// TIA Portal V19 export
FUNCTION_BLOCK "HU_Tank"   // FB107, LAD
TITLE = Hydraulic Tank Machine / HYDRAULIC UNIT (MONO-PUMP)
// stored: Access Published, MemoryReserve 100, SetENOAutomatically false
   VAR_INPUT
      AreaInterface : "AreaInterface";
      DataIn : Struct
         SensorLevelOk_Warning : Bool;
         SensorLevelOk_Alarm : Bool;
         SensorOilMaxTempOk : Bool;
         SensorRecircFilterClogged : Bool;
         SwThermostatCooling : Bool;
         RecircPump_FdbkRunning : Bool;
         HeatExchangeFan_FdbkRunning : Bool;
         HeatingUnit1_FdbkRunning : Bool;
         HeatingUnit2_FdbkRunning : Bool;
         ChillerWaterFluxOk : Bool;
         ChillerAlarmPresence : Bool;
         Anl_OilTemperature : Int;
         Anl_WaterTemperature : Int;
      END_STRUCT;
      CIn : Struct
         PumpRunning : Bool;   // From HU_Pump
      END_STRUCT;
      Config : "HU_Tank_Config";
      Simulation : Bool;
   END_VAR
   VAR_OUTPUT
      MachineInterface : "MachineInterface";
      DataOut : Struct
         KmHeatExchangerFan : Bool;
         KmRecirculationPump : Bool;
         KmHeatingUnit1 : Bool;
         KmHeatingUnit2 : Bool;
         EvChillerWater : Bool;
      END_STRUCT;
      COut : Struct
         PumpRunPermitted : Bool;   // For HU_Pump
         EnableCheckFIler : Bool;   // For HU_Pump
      END_STRUCT;
   END_VAR
   VAR_IN_OUT
      Par : "HU_Tank_Par";
   END_VAR
   VAR
      M_RecirculationPump : "Motor";
      M_HeatExchangerFan : "Motor";
      M_HeatingUnit1 : "Motor";
      M_HeatingUnit2 : "Motor";
      Ctrl : Struct
         RstAlarms : Bool;
         RecirculationPump_Run : Bool;
         HeatExchangerFan_Run : Bool;
         HeatingUnit1_Run : Bool;
         HeatingUnit2_Run : Bool;
      END_STRUCT;
      Sts : Struct
         AlarmsPresence : Bool;
         WarningsPresence : Bool;
         IsStandstill : Bool;
         CoolingReq : Bool;
         HeatingReq : Bool;
         CndRecirculationPump : Bool;
         CndHeatExchangerFan : Bool;
         CndHeatingUnit : Bool;
         OilMaxTemperature : Bool;
         FilterWatchEnableByTemperature : Bool;
         WeeklyClockEnabled : Bool;
         OilTemperature : Real;
         WaterTemperature : Real;
      END_STRUCT;
      HMI : "HU_Tank_HMI";
      Alarm : Struct
         LowTankLevel : Bool;
         OilMaxTemperature : Bool;
         RecircFilterClogged : Bool;
         RecirculationPump : "MotorAlr";
         HeatExchangerFan : "MotorAlr";
         HeatingUnit1 : "MotorAlr";
         HeatingUnit2 : "MotorAlr";
      END_STRUCT;
      Warning : Struct
         NoAutReady : Bool;
         LowTankLevel : Bool;
         CoolingActive : Bool;
         HeatingActive : Bool;
         ChillerLowWater : Bool;
         ChillerAlarm : Bool;
         ChillerWaterMaxTemp : Bool;
         WaitingStartCondition : Bool;
      END_STRUCT;
      tonLowLevel_Warning : IEC_TIMER;
      tonLowLevel_Alarm : IEC_TIMER;
      tonOilMaxTemperature : IEC_TIMER;
      tonAlrRecircFilterClogged : IEC_TIMER;
      tonRecirculationPumpStop : IEC_TIMER;
      tonCoolingStop : IEC_TIMER;
      tonCoolingStart : IEC_TIMER;
      tonDelayCheckChiller : IEC_TIMER;
      tonDelayStartHeating1 : IEC_TIMER;
      tonDelayStopHeating1 : IEC_TIMER;
      tonDelayStartHeating2 : IEC_TIMER;
      tonDelayStopHeating2 : IEC_TIMER;
   END_VAR
   VAR DB_SPECIFIC
      ActualDT : DTL;
      ActualDate : Date;
      ActuaDtON : DTL;
      ActualDtOFF : DTL;
   END_VAR
   VAR
      AckRstAlarms : Bool;
   END_VAR
   VAR_TEMP
      ScaleRetVal : Word;
      StartHeating : Real;
      StopHeating : Real;
      DateRetVal : Int;
      IsGt : Bool;
      IsLt : Bool;
   END_VAR
BEGIN

REGION Network 1 (SCL): Info
   //=============================================================================
   //PM FORMING
   //-----------------------------------------------------------------------------
   // Library: StandardBlocks
   // Tested with: S7-1518TF
   // Engineering: TIA Portal V18
   // Restrictions: -
   // Requirements: S7-1500
   // Functionality: Hydraulic Tank Machine
   //
   // v1.0.0  28/12/2022 
   // v1.0.1  16/01/2023 Added Weekly clock
   // v1.1.0  14/02/2023 Simulation added
   // v1.1.1  11/05/2023 Added config analogic High and low limit
   // v1.1.2  14/06/2023 Set Sensor filter clogged NO
   // v1.1.3  13/11/2023 Add recirculation pump not exist for heating condition
   // v1.1.4  05/03/2024 Add condition low level for recirculation and heating unit
   // v1.1.5  29/04/2024 Add reset filter clogged
   //=============================================================================
END_REGION

REGION Network 2 (SCL): Reset alarms command
   #Ctrl.RstAlarms := #AreaInterface.RstAlarms AND NOT #AckRstAlarms;
   #AckRstAlarms := #AreaInterface.RstAlarms;

   IF #Ctrl.RstAlarms THEN
       #Warning.NoAutReady := FALSE;
       #Alarm.LowTankLevel :=  FALSE;
       #Alarm.OilMaxTemperature := FALSE;    
       #Alarm.RecircFilterClogged := FALSE;
   END_IF;
END_REGION

REGION Network 3: Warning low level
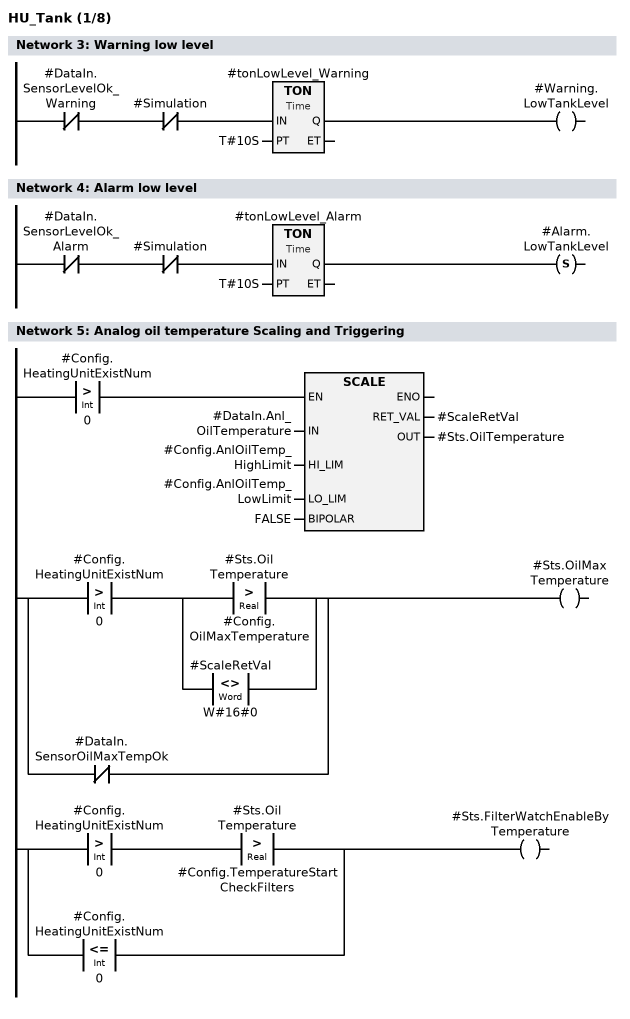
   RUNG wire#powerrail
      I_Contact( #DataIn.SensorLevelOk_Warning )
      I_Contact( #Simulation )
      { S7_Templates := "time_type := Time" } #tonLowLevel_Warning.TON(pt := T#10S, et =>)
      Coil( #Warning.LowTankLevel )
   END_RUNG
   // the same network as SCL:
   #tonLowLevel_Warning.TON(IN := NOT #DataIn.SensorLevelOk_Warning AND NOT #Simulation, PT := T#10S);
   #Warning.LowTankLevel := #tonLowLevel_Warning.Q;
END_REGION

REGION Network 4: Alarm low level
   RUNG wire#powerrail
      I_Contact( #DataIn.SensorLevelOk_Alarm )
      I_Contact( #Simulation )
      { S7_Templates := "time_type := Time" } #tonLowLevel_Alarm.TON(pt := T#10S, et =>)
      S_Coil( #Alarm.LowTankLevel )
   END_RUNG
   // the same network as SCL:
   #tonLowLevel_Alarm.TON(IN := NOT #DataIn.SensorLevelOk_Alarm AND NOT #Simulation, PT := T#10S);
   IF #tonLowLevel_Alarm.Q THEN #Alarm.LowTankLevel := TRUE; END_IF;
END_REGION

REGION Network 5: Analog oil temperature Scaling and Triggering
   IF #Config.HeatingUnitExistNum > 0 THEN
       #ScaleRetVal := SCALE(IN := #DataIn.Anl_OilTemperature,
                             HI_LIM := #Config.AnlOilTemp_HighLimit,
                             LO_LIM := #Config.AnlOilTemp_LowLimit,
                             BIPOLAR := FALSE,
                             OUT => #Sts.OilTemperature);
   END_IF;
   #Sts.OilMaxTemperature := ((#Config.HeatingUnitExistNum > 0) AND ((#Sts.OilTemperature > #Config.OilMaxTemperature) OR (#ScaleRetVal <> W#16#0))) OR NOT #DataIn.SensorOilMaxTempOk;
   #Sts.FilterWatchEnableByTemperature := ((#Config.HeatingUnitExistNum > 0) AND (#Sts.OilTemperature > #Config.TemperatureStartCheckFilters)) OR (#Config.HeatingUnitExistNum <= 0);
END_REGION

REGION Network 6: Analog water temperature Scaling and Triggering
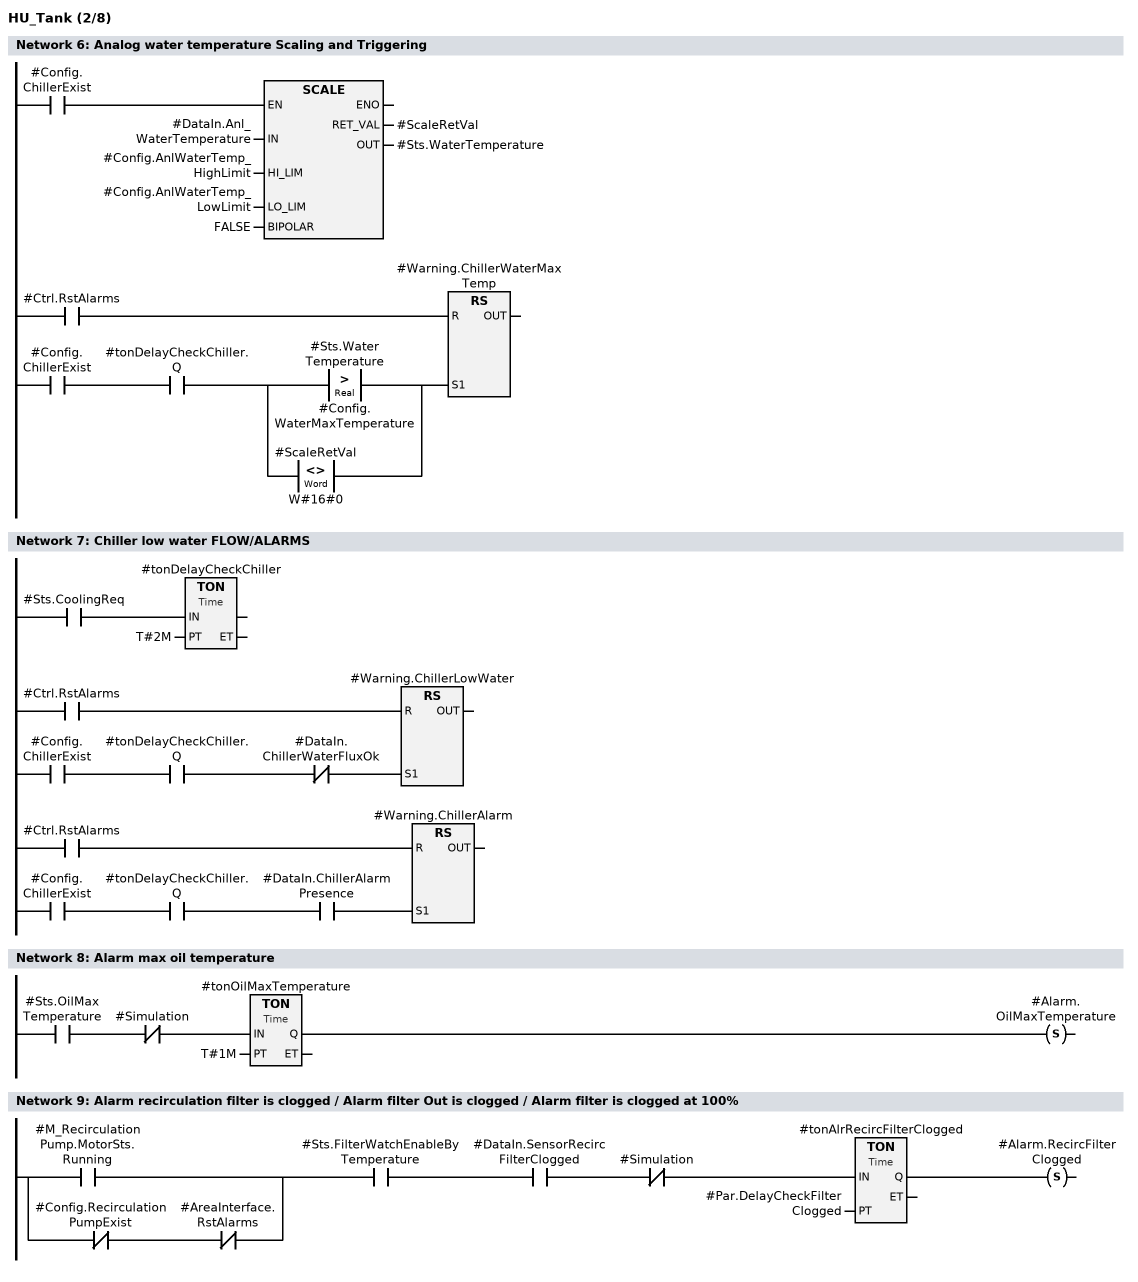
   IF #Config.ChillerExist THEN
       #ScaleRetVal := SCALE(IN := #DataIn.Anl_WaterTemperature,
                             HI_LIM := #Config.AnlWaterTemp_HighLimit,
                             LO_LIM := #Config.AnlWaterTemp_LowLimit,
                             BIPOLAR := FALSE,
                             OUT => #Sts.WaterTemperature);
   END_IF;
   IF #Ctrl.RstAlarms THEN
       #Warning.ChillerWaterMaxTemp := FALSE;   // RS flip-flop
   END_IF;
   IF #Config.ChillerExist AND #tonDelayCheckChiller.Q AND ((#Sts.WaterTemperature > #Config.WaterMaxTemperature) OR (#ScaleRetVal <> W#16#0)) THEN
       #Warning.ChillerWaterMaxTemp := TRUE;
   END_IF;
END_REGION

REGION Network 7: Chiller low water FLOW/ALARMS
   RUNG wire#powerrail
      Contact( #Sts.CoolingReq )
      { S7_Templates := "time_type := Time" } #tonDelayCheckChiller.TON(pt := T#2M, et =>)
   END_RUNG
   RUNG wire#powerrail
      Contact( #Ctrl.RstAlarms )
      S_RS(operand := #Warning.ChillerLowWater, s1 := wire#w1)
   END_RUNG
   RUNG wire#powerrail
      Contact( #Config.ChillerExist )
      Contact( #tonDelayCheckChiller.Q )
      I_Contact( #DataIn.ChillerWaterFluxOk )
   END_RUNG wire#w1
   RUNG wire#powerrail
      Contact( #Ctrl.RstAlarms )
      S_RS(operand := #Warning.ChillerAlarm, s1 := wire#w2)
   END_RUNG
   RUNG wire#powerrail
      Contact( #Config.ChillerExist )
      Contact( #tonDelayCheckChiller.Q )
      Contact( #DataIn.ChillerAlarmPresence )
   END_RUNG wire#w2
   // the same network as SCL:
   #tonDelayCheckChiller.TON(IN := #Sts.CoolingReq, PT := T#2M);
   IF #Ctrl.RstAlarms THEN
       #Warning.ChillerLowWater := FALSE;   // RS flip-flop
   END_IF;
   IF #Config.ChillerExist AND #tonDelayCheckChiller.Q AND NOT #DataIn.ChillerWaterFluxOk THEN
       #Warning.ChillerLowWater := TRUE;
   END_IF;
   IF #Ctrl.RstAlarms THEN
       #Warning.ChillerAlarm := FALSE;   // RS flip-flop
   END_IF;
   IF #Config.ChillerExist AND #tonDelayCheckChiller.Q AND #DataIn.ChillerAlarmPresence THEN
       #Warning.ChillerAlarm := TRUE;
   END_IF;
END_REGION

REGION Network 8: Alarm max oil temperature
   RUNG wire#powerrail
      Contact( #Sts.OilMaxTemperature )
      I_Contact( #Simulation )
      { S7_Templates := "time_type := Time" } #tonOilMaxTemperature.TON(pt := T#1M, et =>)
      S_Coil( #Alarm.OilMaxTemperature )
   END_RUNG
   // the same network as SCL:
   #tonOilMaxTemperature.TON(IN := #Sts.OilMaxTemperature AND NOT #Simulation, PT := T#1M);
   IF #tonOilMaxTemperature.Q THEN #Alarm.OilMaxTemperature := TRUE; END_IF;
END_REGION

REGION Network 9: Alarm recirculation filter is clogged / Alarm filter Out is clogged / Alarm filter is clogged at 100%
   RUNG wire#powerrail
      Contact( #M_RecirculationPump.MotorSts.Running )
      wire#w1
      Contact( #Sts.FilterWatchEnableByTemperature )
      Contact( #DataIn.SensorRecircFilterClogged )
      I_Contact( #Simulation )
      { S7_Templates := "time_type := Time" } #tonAlrRecircFilterClogged.TON(pt := #Par.DelayCheckFilterClogged, et =>)
      S_Coil( #Alarm.RecircFilterClogged )
   END_RUNG
   RUNG wire#powerrail
      I_Contact( #Config.RecirculationPumpExist )
      I_Contact( #AreaInterface.RstAlarms )
   END_RUNG wire#w1
   // the same network as SCL:
   #tonAlrRecircFilterClogged.TON(IN := (#M_RecirculationPump.MotorSts.Running OR (NOT #Config.RecirculationPumpExist AND NOT #AreaInterface.RstAlarms)) AND #Sts.FilterWatchEnableByTemperature AND #DataIn.SensorRecircFilterClogged AND NOT #Simulation,
                           PT := #Par.DelayCheckFilterClogged);
   IF #tonAlrRecircFilterClogged.Q THEN #Alarm.RecircFilterClogged := TRUE; END_IF;
END_REGION

REGION Network 11: <<< HEAT EXCHANGER (RECIRCULATION PUMP & COOLING FAN) / <<< RECIRCULATION PUMP & COOLING FAN >>>
END_REGION

REGION Network 12: Main / Cooling request / Cooling request by thermostat
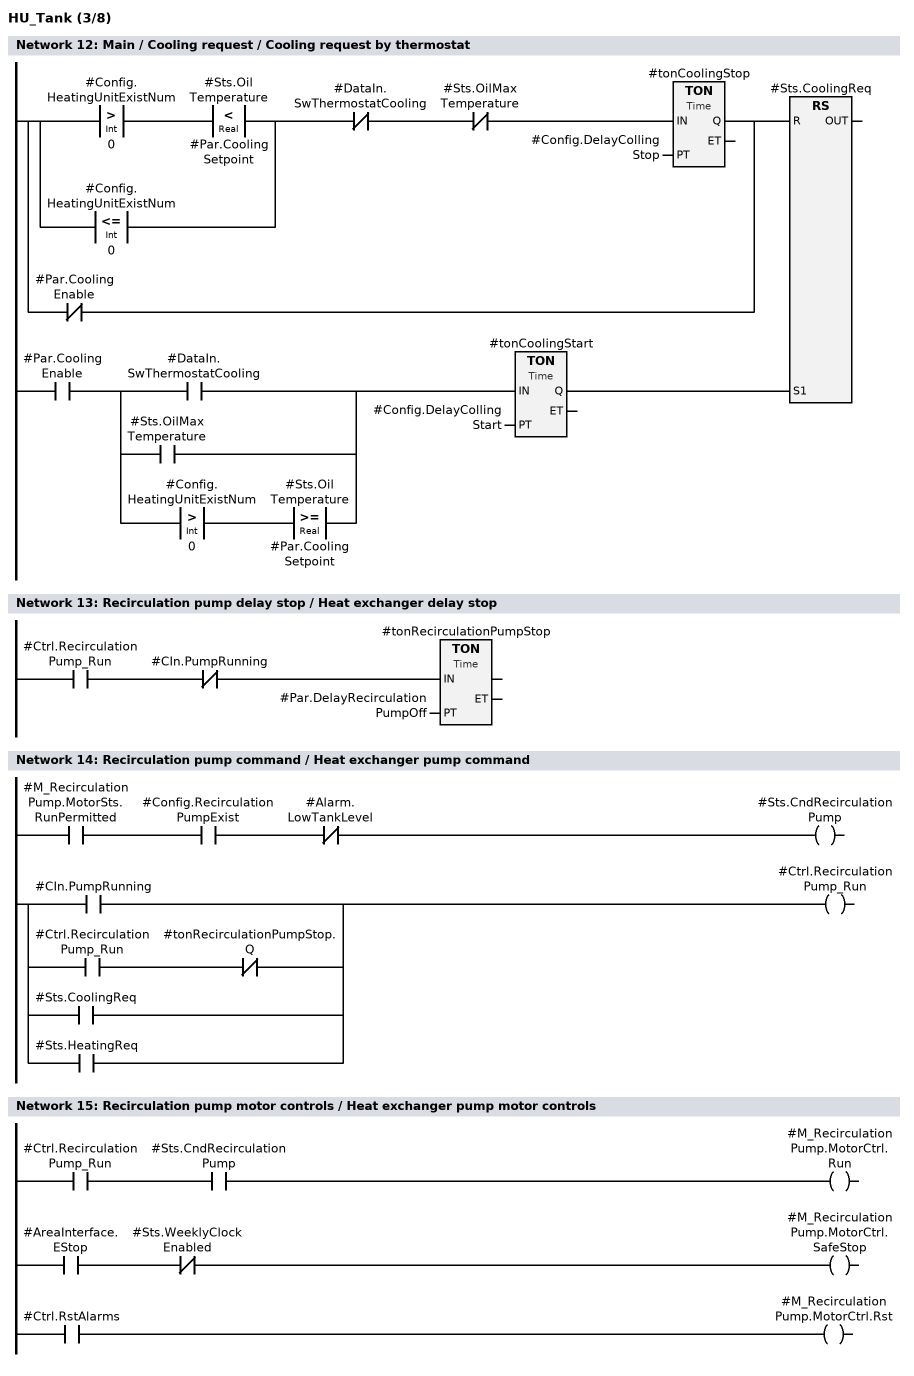
   RUNG wire#powerrail
      { S7_Templates := "SrcType := Int" } GT_Contact(in1 := #Config.HeatingUnitExistNum, in2 := 0)
      { S7_Templates := "SrcType := Real" } LT_Contact(in1 := #Sts.OilTemperature, in2 := #Par.CoolingSetpoint)
      wire#w1
      I_Contact( #DataIn.SwThermostatCooling )
      I_Contact( #Sts.OilMaxTemperature )
      { S7_Templates := "time_type := Time" } #tonCoolingStop.TON(pt := #Config.DelayCollingStop, et =>)
      wire#w2
      S_RS(operand := #Sts.CoolingReq, s1 := wire#w5)
   END_RUNG
   RUNG wire#powerrail
      { S7_Templates := "SrcType := Int" } LE_Contact(in1 := #Config.HeatingUnitExistNum, in2 := 0)
   END_RUNG wire#w1
   RUNG wire#powerrail
      I_Contact( #Par.CoolingEnable )
   END_RUNG wire#w2
   RUNG wire#powerrail
      Contact( #Par.CoolingEnable )
      wire#w3
      Contact( #DataIn.SwThermostatCooling )
      wire#w4
      { S7_Templates := "time_type := Time" } #tonCoolingStart.TON(pt := #Config.DelayCollingStart, et =>)
   END_RUNG wire#w5
   RUNG wire#w3
      Contact( #Sts.OilMaxTemperature )
   END_RUNG wire#w4
   RUNG wire#w3
      { S7_Templates := "SrcType := Int" } GT_Contact(in1 := #Config.HeatingUnitExistNum, in2 := 0)
      { S7_Templates := "SrcType := Real" } GE_Contact(in1 := #Sts.OilTemperature, in2 := #Par.CoolingSetpoint)
   END_RUNG wire#w4
   // the same network as SCL:
   #tonCoolingStop.TON(IN := (((#Config.HeatingUnitExistNum > 0) AND (#Sts.OilTemperature < #Par.CoolingSetpoint)) OR (#Config.HeatingUnitExistNum <= 0)) AND NOT #DataIn.SwThermostatCooling AND NOT #Sts.OilMaxTemperature,
                       PT := #Config.DelayCollingStop);
   #tonCoolingStart.TON(IN := #Par.CoolingEnable AND (#DataIn.SwThermostatCooling OR #Sts.OilMaxTemperature OR ((#Config.HeatingUnitExistNum > 0) AND (#Sts.OilTemperature >= #Par.CoolingSetpoint))),
                        PT := #Config.DelayCollingStart);
   IF #tonCoolingStop.Q OR NOT #Par.CoolingEnable THEN
       #Sts.CoolingReq := FALSE;   // RS flip-flop
   END_IF;
   IF #tonCoolingStart.Q THEN #Sts.CoolingReq := TRUE; END_IF;
END_REGION

REGION Network 13: Recirculation pump delay stop / Heat exchanger delay stop
   RUNG wire#powerrail
      Contact( #Ctrl.RecirculationPump_Run )
      I_Contact( #CIn.PumpRunning )
      { S7_Templates := "time_type := Time" } #tonRecirculationPumpStop.TON(pt := #Par.DelayRecirculationPumpOff, et =>)
   END_RUNG
   // the same network as SCL:
   #tonRecirculationPumpStop.TON(IN := #Ctrl.RecirculationPump_Run AND NOT #CIn.PumpRunning,
                           PT := #Par.DelayRecirculationPumpOff);
END_REGION

REGION Network 14: Recirculation pump command / Heat exchanger pump command
   RUNG wire#powerrail
      Contact( #M_RecirculationPump.MotorSts.RunPermitted )
      Contact( #Config.RecirculationPumpExist )
      I_Contact( #Alarm.LowTankLevel )
      Coil( #Sts.CndRecirculationPump )
   END_RUNG
   RUNG wire#powerrail
      Contact( #CIn.PumpRunning )
      wire#w1
      Coil( #Ctrl.RecirculationPump_Run )
   END_RUNG
   RUNG wire#powerrail
      Contact( #Ctrl.RecirculationPump_Run )
      I_Contact( #tonRecirculationPumpStop.Q )
   END_RUNG wire#w1
   RUNG wire#powerrail
      Contact( #Sts.CoolingReq )
   END_RUNG wire#w1
   RUNG wire#powerrail
      Contact( #Sts.HeatingReq )
   END_RUNG wire#w1
   // the same network as SCL:
   #Sts.CndRecirculationPump := #M_RecirculationPump.MotorSts.RunPermitted AND #Config.RecirculationPumpExist AND NOT #Alarm.LowTankLevel;
   #Ctrl.RecirculationPump_Run := #CIn.PumpRunning OR (#Ctrl.RecirculationPump_Run AND NOT #tonRecirculationPumpStop.Q) OR #Sts.CoolingReq OR #Sts.HeatingReq;
END_REGION

REGION Network 15: Recirculation pump motor controls / Heat exchanger pump motor controls
   RUNG wire#powerrail
      Contact( #Ctrl.RecirculationPump_Run )
      Contact( #Sts.CndRecirculationPump )
      Coil( #M_RecirculationPump.MotorCtrl.Run )
   END_RUNG
   RUNG wire#powerrail
      Contact( #AreaInterface.EStop )
      I_Contact( #Sts.WeeklyClockEnabled )
      Coil( #M_RecirculationPump.MotorCtrl.SafeStop )
   END_RUNG
   RUNG wire#powerrail
      Contact( #Ctrl.RstAlarms )
      Coil( #M_RecirculationPump.MotorCtrl.Rst )
   END_RUNG
   // the same network as SCL:
   #M_RecirculationPump.MotorCtrl.Run := #Ctrl.RecirculationPump_Run AND #Sts.CndRecirculationPump;
   #M_RecirculationPump.MotorCtrl.SafeStop := #AreaInterface.EStop AND NOT #Sts.WeeklyClockEnabled;
   #M_RecirculationPump.MotorCtrl.Rst := #Ctrl.RstAlarms;
END_REGION

REGION Network 16: Recirculation pump motor manager / Heat exchanger pump motor manager
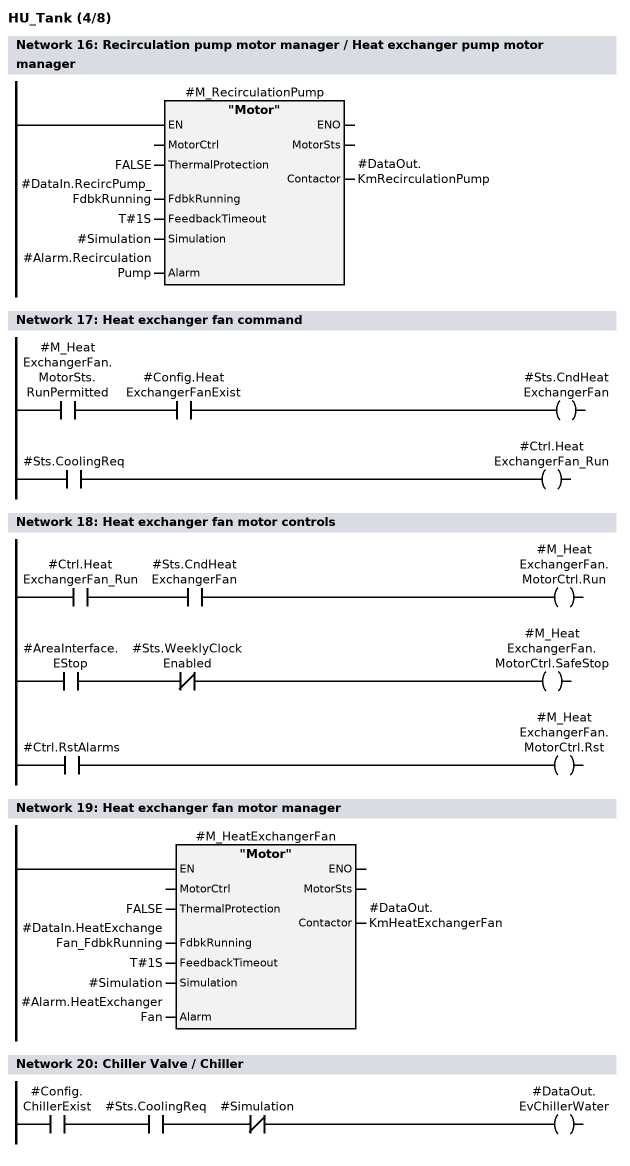
   RUNG wire#powerrail
      #M_RecirculationPump(MotorCtrl :=, ThermalProtection := FALSE, FdbkRunning := #DataIn.RecircPump_FdbkRunning, FeedbackTimeout := T#1S, Simulation := #Simulation, Alarm := #Alarm.RecirculationPump, MotorSts =>, Contactor => #DataOut.KmRecirculationPump)
   END_RUNG
   // the same network as SCL:
   #M_RecirculationPump(ThermalProtection := FALSE,   // "Motor"
                        FdbkRunning := #DataIn.RecircPump_FdbkRunning,
                        FeedbackTimeout := T#1S,
                        Simulation := #Simulation,
                        Alarm := #Alarm.RecirculationPump,
                        Contactor => #DataOut.KmRecirculationPump);
END_REGION

REGION Network 17: Heat exchanger fan command
   RUNG wire#powerrail
      Contact( #M_HeatExchangerFan.MotorSts.RunPermitted )
      Contact( #Config.HeatExchangerFanExist )
      Coil( #Sts.CndHeatExchangerFan )
   END_RUNG
   RUNG wire#powerrail
      Contact( #Sts.CoolingReq )
      Coil( #Ctrl.HeatExchangerFan_Run )
   END_RUNG
   // the same network as SCL:
   #Sts.CndHeatExchangerFan := #M_HeatExchangerFan.MotorSts.RunPermitted AND #Config.HeatExchangerFanExist;
   #Ctrl.HeatExchangerFan_Run := #Sts.CoolingReq;
END_REGION

REGION Network 18: Heat exchanger fan motor controls
   RUNG wire#powerrail
      Contact( #Ctrl.HeatExchangerFan_Run )
      Contact( #Sts.CndHeatExchangerFan )
      Coil( #M_HeatExchangerFan.MotorCtrl.Run )
   END_RUNG
   RUNG wire#powerrail
      Contact( #AreaInterface.EStop )
      I_Contact( #Sts.WeeklyClockEnabled )
      Coil( #M_HeatExchangerFan.MotorCtrl.SafeStop )
   END_RUNG
   RUNG wire#powerrail
      Contact( #Ctrl.RstAlarms )
      Coil( #M_HeatExchangerFan.MotorCtrl.Rst )
   END_RUNG
   // the same network as SCL:
   #M_HeatExchangerFan.MotorCtrl.Run := #Ctrl.HeatExchangerFan_Run AND #Sts.CndHeatExchangerFan;
   #M_HeatExchangerFan.MotorCtrl.SafeStop := #AreaInterface.EStop AND NOT #Sts.WeeklyClockEnabled;
   #M_HeatExchangerFan.MotorCtrl.Rst := #Ctrl.RstAlarms;
END_REGION

REGION Network 19: Heat exchanger fan motor manager
   RUNG wire#powerrail
      #M_HeatExchangerFan(MotorCtrl :=, ThermalProtection := FALSE, FdbkRunning := #DataIn.HeatExchangeFan_FdbkRunning, FeedbackTimeout := T#1S, Simulation := #Simulation, Alarm := #Alarm.HeatExchangerFan, MotorSts =>, Contactor => #DataOut.KmHeatExchangerFan)
   END_RUNG
   // the same network as SCL:
   #M_HeatExchangerFan(ThermalProtection := FALSE,   // "Motor"
                       FdbkRunning := #DataIn.HeatExchangeFan_FdbkRunning,
                       FeedbackTimeout := T#1S,
                       Simulation := #Simulation,
                       Alarm := #Alarm.HeatExchangerFan,
                       Contactor => #DataOut.KmHeatExchangerFan);
END_REGION

REGION Network 20: Chiller Valve / Chiller
   RUNG wire#powerrail
      Contact( #Config.ChillerExist )
      Contact( #Sts.CoolingReq )
      I_Contact( #Simulation )
      Coil( #DataOut.EvChillerWater )
   END_RUNG
   // the same network as SCL:
   #DataOut.EvChillerWater := #Config.ChillerExist AND #Sts.CoolingReq AND NOT #Simulation;
END_REGION

REGION Network 22: <<< HEATING >>>
END_REGION

REGION Network 23: Main
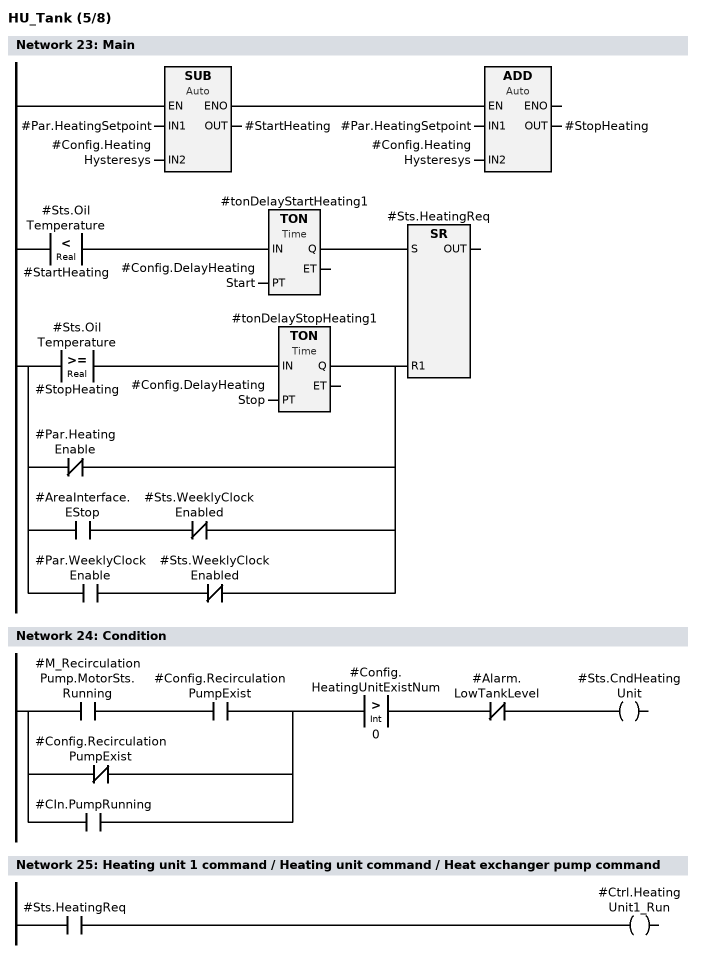
   RUNG wire#powerrail
      Sub(in1 := #Par.HeatingSetpoint, in2 := #Config.HeatingHysteresys, out => #StartHeating)
      Add(in1 := #Par.HeatingSetpoint, in2 := #Config.HeatingHysteresys, out => #StopHeating)
   END_RUNG
   RUNG wire#powerrail
      { S7_Templates := "SrcType := Real" } LT_Contact(in1 := #Sts.OilTemperature, in2 := #StartHeating)
      { S7_Templates := "time_type := Time" } #tonDelayStartHeating1.TON(pt := #Config.DelayHeatingStart, et =>)
      S_SR(operand := #Sts.HeatingReq, r1 := wire#w1)
   END_RUNG
   RUNG wire#powerrail
      { S7_Templates := "SrcType := Real" } GE_Contact(in1 := #Sts.OilTemperature, in2 := #StopHeating)
      { S7_Templates := "time_type := Time" } #tonDelayStopHeating1.TON(pt := #Config.DelayHeatingStop, et =>)
   END_RUNG wire#w1
   RUNG wire#powerrail
      I_Contact( #Par.HeatingEnable )
   END_RUNG wire#w1
   RUNG wire#powerrail
      Contact( #AreaInterface.EStop )
      I_Contact( #Sts.WeeklyClockEnabled )
   END_RUNG wire#w1
   RUNG wire#powerrail
      Contact( #Par.WeeklyClockEnable )
      I_Contact( #Sts.WeeklyClockEnabled )
   END_RUNG wire#w1
   // the same network as SCL:
   #StartHeating := #Par.HeatingSetpoint - #Config.HeatingHysteresys;
   #StopHeating := #Par.HeatingSetpoint + #Config.HeatingHysteresys;
   #tonDelayStartHeating1.TON(IN := #Sts.OilTemperature < #StartHeating, PT := #Config.DelayHeatingStart);
   #tonDelayStopHeating1.TON(IN := #Sts.OilTemperature >= #StopHeating, PT := #Config.DelayHeatingStop);
   IF #tonDelayStartHeating1.Q THEN
       #Sts.HeatingReq := TRUE;   // SR flip-flop
   END_IF;
   IF #tonDelayStopHeating1.Q OR NOT #Par.HeatingEnable OR (#AreaInterface.EStop AND NOT #Sts.WeeklyClockEnabled) OR (#Par.WeeklyClockEnable AND NOT #Sts.WeeklyClockEnabled) THEN
       #Sts.HeatingReq := FALSE;
   END_IF;
END_REGION

REGION Network 24: Condition
   RUNG wire#powerrail
      Contact( #M_RecirculationPump.MotorSts.Running )
      Contact( #Config.RecirculationPumpExist )
      wire#w1
      { S7_Templates := "SrcType := Int" } GT_Contact(in1 := #Config.HeatingUnitExistNum, in2 := 0)
      I_Contact( #Alarm.LowTankLevel )
      Coil( #Sts.CndHeatingUnit )
   END_RUNG
   RUNG wire#powerrail
      I_Contact( #Config.RecirculationPumpExist )
   END_RUNG wire#w1
   RUNG wire#powerrail
      Contact( #CIn.PumpRunning )
   END_RUNG wire#w1
   // the same network as SCL:
   #Sts.CndHeatingUnit := ((#M_RecirculationPump.MotorSts.Running AND #Config.RecirculationPumpExist) OR NOT #Config.RecirculationPumpExist OR #CIn.PumpRunning) AND (#Config.HeatingUnitExistNum > 0) AND NOT #Alarm.LowTankLevel;
END_REGION

REGION Network 25: Heating unit 1 command / Heating unit command / Heat exchanger pump command
   RUNG wire#powerrail
      Contact( #Sts.HeatingReq )
      Coil( #Ctrl.HeatingUnit1_Run )
   END_RUNG
   // the same network as SCL:
   #Ctrl.HeatingUnit1_Run := #Sts.HeatingReq;
END_REGION

REGION Network 26: Heating unit 2 command
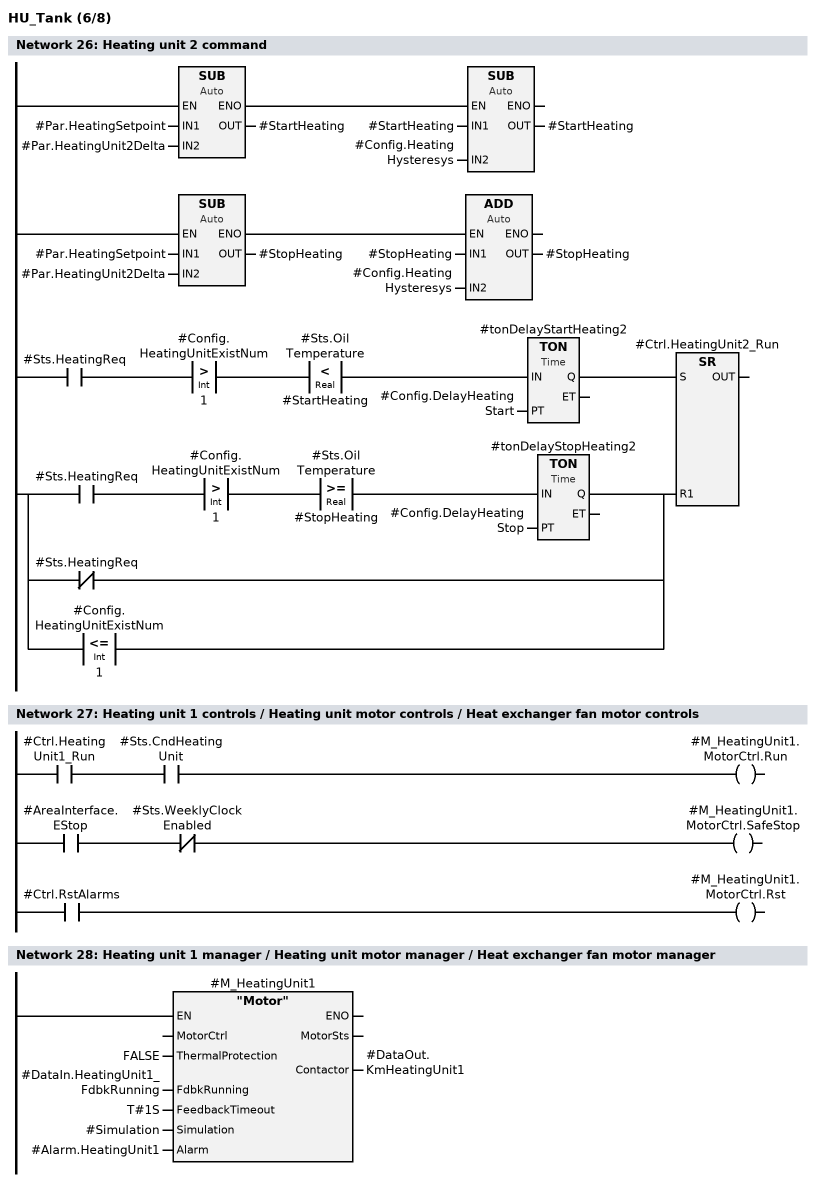
   RUNG wire#powerrail
      Sub(in1 := #Par.HeatingSetpoint, in2 := #Par.HeatingUnit2Delta, out => #StartHeating)
      Sub(in1 := #StartHeating, in2 := #Config.HeatingHysteresys, out => #StartHeating)
   END_RUNG
   RUNG wire#powerrail
      Sub(in1 := #Par.HeatingSetpoint, in2 := #Par.HeatingUnit2Delta, out => #StopHeating)
      Add(in1 := #StopHeating, in2 := #Config.HeatingHysteresys, out => #StopHeating)
   END_RUNG
   RUNG wire#powerrail
      Contact( #Sts.HeatingReq )
      { S7_Templates := "SrcType := Int" } GT_Contact(in1 := #Config.HeatingUnitExistNum, in2 := 1)
      { S7_Templates := "SrcType := Real" } LT_Contact(in1 := #Sts.OilTemperature, in2 := #StartHeating)
      { S7_Templates := "time_type := Time" } #tonDelayStartHeating2.TON(pt := #Config.DelayHeatingStart, et =>)
      S_SR(operand := #Ctrl.HeatingUnit2_Run, r1 := wire#w1)
   END_RUNG
   RUNG wire#powerrail
      Contact( #Sts.HeatingReq )
      { S7_Templates := "SrcType := Int" } GT_Contact(in1 := #Config.HeatingUnitExistNum, in2 := 1)
      { S7_Templates := "SrcType := Real" } GE_Contact(in1 := #Sts.OilTemperature, in2 := #StopHeating)
      { S7_Templates := "time_type := Time" } #tonDelayStopHeating2.TON(pt := #Config.DelayHeatingStop, et =>)
   END_RUNG wire#w1
   RUNG wire#powerrail
      I_Contact( #Sts.HeatingReq )
   END_RUNG wire#w1
   RUNG wire#powerrail
      { S7_Templates := "SrcType := Int" } LE_Contact(in1 := #Config.HeatingUnitExistNum, in2 := 1)
   END_RUNG wire#w1
   // the same network as SCL:
   #StartHeating := #Par.HeatingSetpoint - #Par.HeatingUnit2Delta;
   #StartHeating := #StartHeating - #Config.HeatingHysteresys;
   #StopHeating := #Par.HeatingSetpoint - #Par.HeatingUnit2Delta;
   #StopHeating := #StopHeating + #Config.HeatingHysteresys;
   #tonDelayStartHeating2.TON(IN := #Sts.HeatingReq AND (#Config.HeatingUnitExistNum > 1) AND (#Sts.OilTemperature < #StartHeating),
                           PT := #Config.DelayHeatingStart);
   #tonDelayStopHeating2.TON(IN := #Sts.HeatingReq AND (#Config.HeatingUnitExistNum > 1) AND (#Sts.OilTemperature >= #StopHeating),
                           PT := #Config.DelayHeatingStop);
   IF #tonDelayStartHeating2.Q THEN
       #Ctrl.HeatingUnit2_Run := TRUE;   // SR flip-flop
   END_IF;
   IF #tonDelayStopHeating2.Q OR NOT #Sts.HeatingReq OR (#Config.HeatingUnitExistNum <= 1) THEN
       #Ctrl.HeatingUnit2_Run := FALSE;
   END_IF;
END_REGION

REGION Network 27: Heating unit 1 controls / Heating unit motor controls / Heat exchanger fan motor controls
   RUNG wire#powerrail
      Contact( #Ctrl.HeatingUnit1_Run )
      Contact( #Sts.CndHeatingUnit )
      Coil( #M_HeatingUnit1.MotorCtrl.Run )
   END_RUNG
   RUNG wire#powerrail
      Contact( #AreaInterface.EStop )
      I_Contact( #Sts.WeeklyClockEnabled )
      Coil( #M_HeatingUnit1.MotorCtrl.SafeStop )
   END_RUNG
   RUNG wire#powerrail
      Contact( #Ctrl.RstAlarms )
      Coil( #M_HeatingUnit1.MotorCtrl.Rst )
   END_RUNG
   // the same network as SCL:
   #M_HeatingUnit1.MotorCtrl.Run := #Ctrl.HeatingUnit1_Run AND #Sts.CndHeatingUnit;
   #M_HeatingUnit1.MotorCtrl.SafeStop := #AreaInterface.EStop AND NOT #Sts.WeeklyClockEnabled;
   #M_HeatingUnit1.MotorCtrl.Rst := #Ctrl.RstAlarms;
END_REGION

REGION Network 28: Heating unit 1 manager / Heating unit motor manager / Heat exchanger fan motor manager
   RUNG wire#powerrail
      #M_HeatingUnit1(MotorCtrl :=, ThermalProtection := FALSE, FdbkRunning := #DataIn.HeatingUnit1_FdbkRunning, FeedbackTimeout := T#1S, Simulation := #Simulation, Alarm := #Alarm.HeatingUnit1, MotorSts =>, Contactor => #DataOut.KmHeatingUnit1)
   END_RUNG
   // the same network as SCL:
   #M_HeatingUnit1(ThermalProtection := FALSE,   // "Motor"
                   FdbkRunning := #DataIn.HeatingUnit1_FdbkRunning,
                   FeedbackTimeout := T#1S,
                   Simulation := #Simulation,
                   Alarm := #Alarm.HeatingUnit1,
                   Contactor => #DataOut.KmHeatingUnit1);
END_REGION

REGION Network 29: Heating unit 2 controls
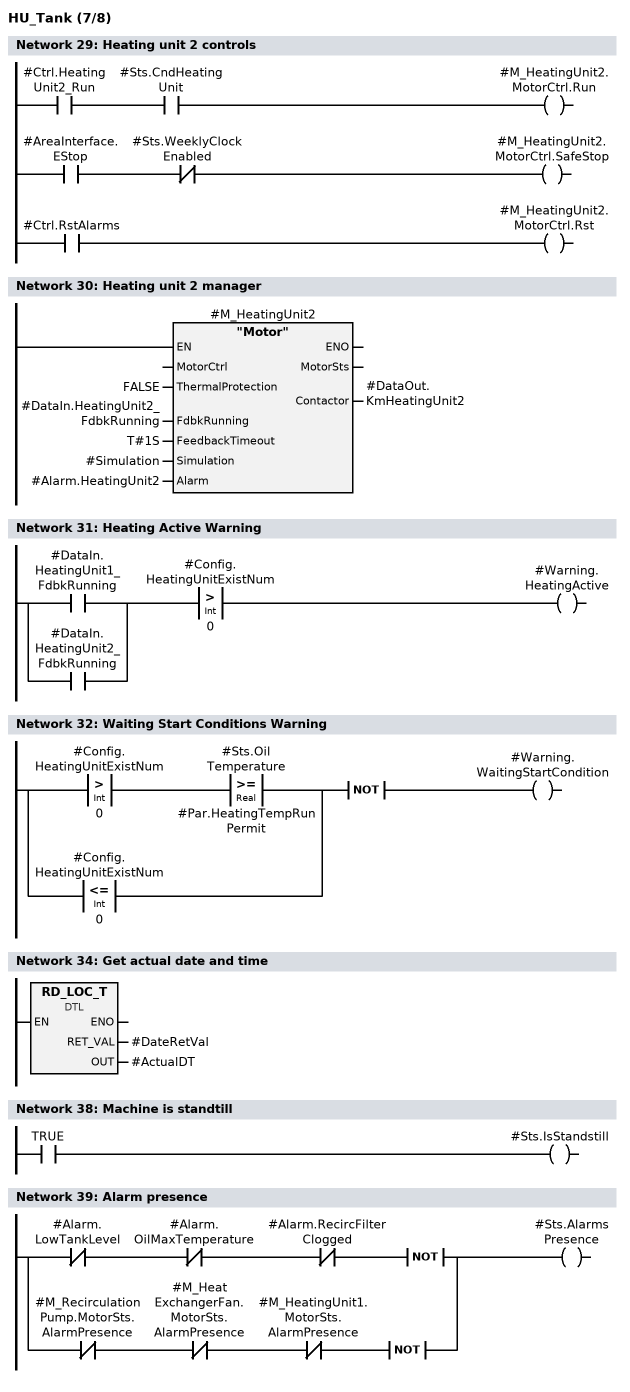
   RUNG wire#powerrail
      Contact( #Ctrl.HeatingUnit2_Run )
      Contact( #Sts.CndHeatingUnit )
      Coil( #M_HeatingUnit2.MotorCtrl.Run )
   END_RUNG
   RUNG wire#powerrail
      Contact( #AreaInterface.EStop )
      I_Contact( #Sts.WeeklyClockEnabled )
      Coil( #M_HeatingUnit2.MotorCtrl.SafeStop )
   END_RUNG
   RUNG wire#powerrail
      Contact( #Ctrl.RstAlarms )
      Coil( #M_HeatingUnit2.MotorCtrl.Rst )
   END_RUNG
   // the same network as SCL:
   #M_HeatingUnit2.MotorCtrl.Run := #Ctrl.HeatingUnit2_Run AND #Sts.CndHeatingUnit;
   #M_HeatingUnit2.MotorCtrl.SafeStop := #AreaInterface.EStop AND NOT #Sts.WeeklyClockEnabled;
   #M_HeatingUnit2.MotorCtrl.Rst := #Ctrl.RstAlarms;
END_REGION

REGION Network 30: Heating unit 2 manager
   RUNG wire#powerrail
      #M_HeatingUnit2(MotorCtrl :=, ThermalProtection := FALSE, FdbkRunning := #DataIn.HeatingUnit2_FdbkRunning, FeedbackTimeout := T#1S, Simulation := #Simulation, Alarm := #Alarm.HeatingUnit2, MotorSts =>, Contactor => #DataOut.KmHeatingUnit2)
   END_RUNG
   // the same network as SCL:
   #M_HeatingUnit2(ThermalProtection := FALSE,   // "Motor"
                   FdbkRunning := #DataIn.HeatingUnit2_FdbkRunning,
                   FeedbackTimeout := T#1S,
                   Simulation := #Simulation,
                   Alarm := #Alarm.HeatingUnit2,
                   Contactor => #DataOut.KmHeatingUnit2);
END_REGION

REGION Network 31: Heating Active Warning
   RUNG wire#powerrail
      Contact( #DataIn.HeatingUnit1_FdbkRunning )
      wire#w1
      { S7_Templates := "SrcType := Int" } GT_Contact(in1 := #Config.HeatingUnitExistNum, in2 := 0)
      Coil( #Warning.HeatingActive )
   END_RUNG
   RUNG wire#powerrail
      Contact( #DataIn.HeatingUnit2_FdbkRunning )
   END_RUNG wire#w1
   // the same network as SCL:
   #Warning.HeatingActive := (#DataIn.HeatingUnit1_FdbkRunning OR #DataIn.HeatingUnit2_FdbkRunning) AND (#Config.HeatingUnitExistNum > 0);
END_REGION

REGION Network 32: Waiting Start Conditions Warning
   RUNG wire#powerrail
      { S7_Templates := "SrcType := Int" } GT_Contact(in1 := #Config.HeatingUnitExistNum, in2 := 0)
      { S7_Templates := "SrcType := Real" } GE_Contact(in1 := #Sts.OilTemperature, in2 := #Par.HeatingTempRunPermit)
      wire#w1
      Not()
      Coil( #Warning.WaitingStartCondition )
   END_RUNG
   RUNG wire#powerrail
      { S7_Templates := "SrcType := Int" } LE_Contact(in1 := #Config.HeatingUnitExistNum, in2 := 0)
   END_RUNG wire#w1
   // the same network as SCL:
   #Warning.WaitingStartCondition := NOT (((#Config.HeatingUnitExistNum > 0) AND (#Sts.OilTemperature >= #Par.HeatingTempRunPermit)) OR (#Config.HeatingUnitExistNum <= 0));
END_REGION

REGION Network 33: <<< WEEKLY CLOCK >>>
END_REGION

REGION Network 34: Get actual date and time
   RUNG wire#powerrail
      { S7_Templates := "date_type := DTL" } RD_LOC_T(RET_VAL => #DateRetVal, OUT => #ActualDT)
   END_RUNG
   // the same network as SCL:
   #DateRetVal := RD_LOC_T(OUT => #ActualDT);
END_REGION

REGION Network 35 (SCL): Days of week for oil Heating
   #ActualDate := DTL_TO_DATE(#ActualDT);
   #ActuaDtON := CONCAT_DATE_TOD(IN1 := #ActualDate, IN2 := #Par.WeeklyClockSetup[#ActualDT.WEEKDAY].Set_ON);
   #ActualDtOFF := CONCAT_DATE_TOD(IN1 := #ActualDate, IN2 :=  #Par.WeeklyClockSetup[#ActualDT.WEEKDAY].Set_OFF);
   #IsGt := #ActualDT >= #ActuaDtON;
   #IsLt := #ActualDT <= #ActualDtOFF;

   #Sts.WeeklyClockEnabled := #IsGt AND #IsLt AND #Par.WeeklyClockSetup[#ActualDT.WEEKDAY].Enable AND #Par.WeeklyClockEnable;
END_REGION

REGION Network 37: <<<< FINAL >>>>>>> / <<<< + >>>>>>>
END_REGION

REGION Network 38: Machine is standtill
   RUNG wire#powerrail
      Contact( TRUE )
      Coil( #Sts.IsStandstill )
   END_RUNG
   // the same network as SCL:
   #Sts.IsStandstill := TRUE;
END_REGION

REGION Network 39: Alarm presence
   RUNG wire#powerrail
      I_Contact( #Alarm.LowTankLevel )
      I_Contact( #Alarm.OilMaxTemperature )
      I_Contact( #Alarm.RecircFilterClogged )
      Not()
      wire#w1
      Coil( #Sts.AlarmsPresence )
   END_RUNG
   RUNG wire#powerrail
      I_Contact( #M_RecirculationPump.MotorSts.AlarmPresence )
      I_Contact( #M_HeatExchangerFan.MotorSts.AlarmPresence )
      I_Contact( #M_HeatingUnit1.MotorSts.AlarmPresence )
      Not()
   END_RUNG wire#w1
   // the same network as SCL:
   #Sts.AlarmsPresence := NOT (NOT #Alarm.LowTankLevel AND NOT #Alarm.OilMaxTemperature AND NOT #Alarm.RecircFilterClogged) OR NOT (NOT #M_RecirculationPump.MotorSts.AlarmPresence AND NOT #M_HeatExchangerFan.MotorSts.AlarmPresence AND NOT #M_HeatingUnit1.MotorSts.AlarmPresence);
END_REGION

REGION Network 40: Warning presence
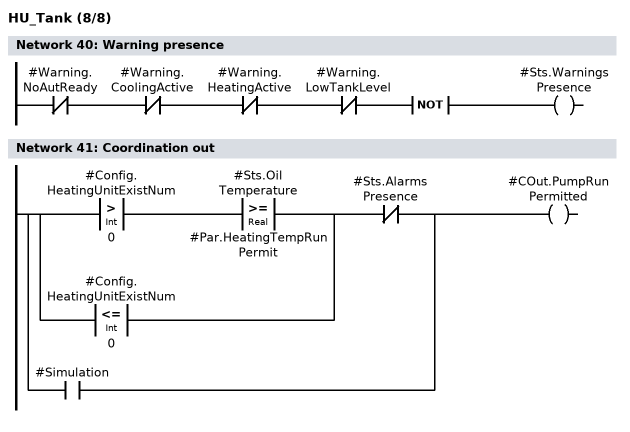
   RUNG wire#powerrail
      I_Contact( #Warning.NoAutReady )
      I_Contact( #Warning.CoolingActive )
      I_Contact( #Warning.HeatingActive )
      I_Contact( #Warning.LowTankLevel )
      Not()
      Coil( #Sts.WarningsPresence )
   END_RUNG
   // the same network as SCL:
   #Sts.WarningsPresence := NOT (NOT #Warning.NoAutReady AND NOT #Warning.CoolingActive AND NOT #Warning.HeatingActive AND NOT #Warning.LowTankLevel);
END_REGION

REGION Network 41: Coordination out
   RUNG wire#powerrail
      { S7_Templates := "SrcType := Int" } GT_Contact(in1 := #Config.HeatingUnitExistNum, in2 := 0)
      { S7_Templates := "SrcType := Real" } GE_Contact(in1 := #Sts.OilTemperature, in2 := #Par.HeatingTempRunPermit)
      wire#w1
      I_Contact( #Sts.AlarmsPresence )
      wire#w2
      Coil( #COut.PumpRunPermitted )
   END_RUNG
   RUNG wire#powerrail
      { S7_Templates := "SrcType := Int" } LE_Contact(in1 := #Config.HeatingUnitExistNum, in2 := 0)
   END_RUNG wire#w1
   RUNG wire#powerrail
      Contact( #Simulation )
   END_RUNG wire#w2
   // the same network as SCL:
   #COut.PumpRunPermitted := ((((#Config.HeatingUnitExistNum > 0) AND (#Sts.OilTemperature >= #Par.HeatingTempRunPermit)) OR (#Config.HeatingUnitExistNum <= 0)) AND NOT #Sts.AlarmsPresence) OR #Simulation;
END_REGION

REGION Network 42 (SCL): HMI
   #HMI.Alarm := #Sts.AlarmsPresence;
   #HMI.RecirculationPump_Running := #M_RecirculationPump.MotorSts.Running;
   #HMI.HeatExchangerFan_Running := #M_HeatExchangerFan.MotorSts.Running;
   #HMI.HeatingUnit1_Running := #M_HeatingUnit1.MotorSts.Running;
   #HMI.HeatingUnit2_Running := #M_HeatingUnit2.MotorSts.Running;
   #HMI.EvChillerWater := #DataOut.EvChillerWater;
   #HMI.OilTemperature := #Sts.OilTemperature;
   #HMI.WaterTemperature := #Sts.WaterTemperature;
END_REGION

REGION Network 43 (SCL): Collect machine to area interface
   // Status machine ready
   #MachineInterface.AutReady := #AreaInterface.Aut AND NOT #Sts.AlarmsPresence;
   // Status machine aborting
   #MachineInterface.Aborting := #Sts.AlarmsPresence;
   // Status Ack Stop in phase
   #MachineInterface.AckStopInPhase :=  #AreaInterface.StopInPhase;
   // Status Ack Stop programmed
   #MachineInterface.AckStopProgrammed := #AreaInterface.StopProgrammed;
   // Status Motion standtill
   #MachineInterface.MotionsStandStill := #Sts.IsStandstill;
   // Status Alarm presence
   #MachineInterface.AlarmsPresence := #Sts.AlarmsPresence;
   // Status Warning presence
   #MachineInterface.WarningPresence := #Sts.WarningsPresence;

   // Warning machine not automatic ready
   IF #AreaInterface.CheckAutReady AND NOT #MachineInterface.AutReady THEN
     #Warning.NoAutReady := false;
   END_IF;
END_REGION
END_FUNCTION_BLOCK
